{attribute 'qualified_only'}
{attribute 'strict'}
TYPE eRxMode :
(
	Delimited	:= 0,
	FixedLength := 1,
	Continuous	:= 2
);
END_TYPE

(* stored: Version 1.1.0.1, ProductVersion 3.1.4024.9
   DUT eRxMode: Id {5dd988c1-3152-4dfc-915e-da4ce43e12a1} *)
